// TIA Portal V20 export
// export: Created 2025-12-01T14:57:45.0435866Z, ExportSetting None, DisplayName Totally Integrated Automation Portal, DisplayVersion V20 Update 3, DisplayName TIA Portal Openness, DisplayVersion V20 Update 3, DisplayName TIA Portal Version Control Interface, DisplayVersion V20 Update 3, DisplayName STEP 7 Professional, DisplayVersion V20 Update 3, DisplayName STEP 7 Safety, DisplayVersion V20 Update 2, DisplayName WinCC Basic/Comfort/Advanced, DisplayVersion V20 Update 3, DisplayName WinCC Professional, DisplayVersion V20 Update 3, DisplayName WinCC Unified, DisplayVersion V20 Update 3
FUNCTION "FC782_Evento_RUES" : Void   // FC782, LAD
{ S7_Optimized_Access := 'FALSE' }
// stored: AutoNumber false, SetENOAutomatically false
   VAR_INPUT
      mensaje : Int;   // indice del array que estamos extrayendo
   END_VAR
   VAR_TEMP
      Existe_ruta : Bool;
      retval : Int;
      pos_SSCC : UInt;
      cero : Byte;
      destinos : Array[0..9] of UInt;
      registro_etiqueta : "ROUT_Reg_Etiqueta";
      orden_desvio : Byte;
      desvio_bits AT orden_desvio : Array[1..8] of Bool;
      posicion : Int;
      pos_ruta : Int;
      posicion_mesa : Int;
      posicion_db : Int;
      desvio : Int;
      scanner : UInt;
      bit_ini : Int;
      n_bits : Int;
      contador_aux : Int;
      contador : Int;
      posicion_BBDD : UInt;
      Atributo_rues : String[4];
   END_VAR
BEGIN

REGION Network 1 (SCL): INICIALIZACIONES
   REGION inicializacion

       // inicializamos las variables
       // 

       #retval := FILL(BVAL := #cero, BLK => #registro_etiqueta); // el registro de la etiqueta temporal
       #retval := FILL(BVAL := #cero, BLK => #destinos); // los datos temporales de los destinos
       #orden_desvio := 0;
       #Existe_ruta := false;

   END_REGION
END_REGION

REGION Network 2 (SCL): EXTRAEMOS DEL MENSAJE LOS DESTINOS

   // miramos si en el mensaje nos han llegado destinos que extraer
   #posicion := FIND(IN1 := "DB199_eventos_convertidos".evento[#mensaje], IN2 := '[DEST]');
   IF #posicion <> 0 THEN    // iniciamos la estracción de las mesas que pertenecen a la ruta
           // si solamente se ejecuta el proceso una vez en el mensaje no es necesario realizar esta operación de sustituir el atributo DEST
       "DB199_eventos_convertidos".evento[#mensaje] := REPLACE(IN1 := "DB199_eventos_convertidos".evento[#mensaje], IN2 := '[dest]', L := 6, P := #posicion);
       #pos_ruta := 0;
       #Existe_ruta := 1;
       // temporalmente ponemos las rutas a cero
       WHILE #Existe_ruta DO
           #posicion := FIND(IN1 := "DB199_eventos_convertidos".evento[#mensaje], IN2 := '[MESA]');
           IF #posicion <> 0 THEN
               STRG_VAL(IN := "DB199_eventos_convertidos".evento[#mensaje],
                        FORMAT := 0,
                        P := (#posicion + 6),
                        OUT => #destinos[#pos_ruta]);
               #pos_ruta += 1; // incrementamos la posición en el array para seguir guardando
               // las mesas ya extraidas, las ponemos en minucula para seguir buscando las siguientes mesas sin eliminar parcialmente el mensaje
               "DB199_eventos_convertidos".evento[#mensaje] := REPLACE(IN1 := "DB199_eventos_convertidos".evento[#mensaje], IN2 := '[mesa]', L := 6, P := #posicion);
           ELSE
               #Existe_ruta := 0;
               EXIT;
           END_IF;
       END_WHILE;
   END_IF;
   // aqui tenemos que incluir la conversión de las mesas el los bits de cruce
END_REGION

REGION Network 3 (SCL): generación de los bits de cruce
   REGION generar_bits_cruce
       #posicion_mesa := 0;
       #posicion_db := 0;

       WHILE #destinos[#posicion_mesa] <> 0 DO
           // Statement section WHILE

           WHILE (("DB913_Router_DestinoDesvio".DestinoDesvios[#posicion_db].Destino <> 0) AND (#posicion_db <= "ROUT_Max_Destinos")) DO
               IF (#destinos[#posicion_mesa] = "DB913_Router_DestinoDesvio".DestinoDesvios[#posicion_db].Destino) THEN
                   // si coincide la mesa con uno de los destinos
                   #desvio := 0;
                   WHILE (("DB913_Router_DestinoDesvio".DestinoDesvios[#posicion_db].Desvios[#desvio].SCR <> 0) AND (#desvio <= "ROUT_Max_Destinos")) DO
                       #scanner := "DB913_Router_DestinoDesvio".DestinoDesvios[#posicion_db].Desvios[#desvio].SCR;
                       #orden_desvio := "DB913_Router_DestinoDesvio".DestinoDesvios[#posicion_db].Desvios[#desvio].Bits;
                       #bit_ini := "DB912_Tipo_Scanner_Router".SCANNER[#scanner].Bit_Ini_Ordenes;
                       #n_bits := "DB912_Tipo_Scanner_Router".SCANNER[#scanner].N_Bits_Orden;

                       // aqui mediante un for vamos escribiendo los bits donde corresponden
                       #contador_aux := 1;
                       FOR #contador := #bit_ini TO (#bit_ini + #n_bits - 1) DO
                           #registro_etiqueta.BIT_Orden[#contador] := #desvio_bits[#contador_aux];
                           #contador_aux += 1;

                       END_FOR;
                       #desvio += 1; // nos desplazamos el siguiente desvio
                   END_WHILE;

               END_IF;
               #posicion_db += 1; //nos desplazamos hasta el siguiente destino
           END_WHILE;
           #posicion_mesa += 1; // nos desplazamos a la siguiente mesa destino de la ruta
           #posicion_db := 0; // inicializamos a cero la busqueda dentro del DB de destinos

       END_WHILE;

   END_REGION
END_REGION

REGION Network 4 (SCL): volcado al DB de datos
   #pos_SSCC := FIND(IN1 := "DB199_eventos_convertidos".evento[#mensaje], IN2 := '[ETES]');
   // extraemos el dato de qué etiqueta especial se trata
   // 

   #Atributo_rues:=MID(IN := "DB199_eventos_convertidos".evento[#mensaje], L := 4, P := (#pos_SSCC + 6));

   // elección de la posición de volcado
   // 
   IF (#Atributo_rues = 'ERRR') THEN
       // especiales registro 1
       "DB209_Reg_Etquetas_Esp_Activa".Reg_Etiqueta[1] := #registro_etiqueta;
   ELSE
       IF (#Atributo_rues = 'NENC') THEN
           // especiales registro 2
           "DB209_Reg_Etquetas_Esp_Activa".Reg_Etiqueta[2] := #registro_etiqueta;
       ELSE
           IF (#Atributo_rues = 'INIC') THEN
               // especiales registro 3
               "DB209_Reg_Etquetas_Esp_Activa".Reg_Etiqueta[3] := #registro_etiqueta;
           END_IF;
       END_IF;
   END_IF;
END_REGION
END_FUNCTION
